# EPICS substitutions: ssaApp/Db/hlCommon.substitutions
# Common controls for cryomodule SSAs.
# Macros:
#   OUT: PV attribute
#   MASK: Bitmask to select which SSAs to control; e.g. 3 for SSAs 1 & 2, 15 for SSAs 1,2,3,4.
#   DLY: Delay between sequence steps

file "ssaCommonControls_4x.template" {
pattern
{       OUT, DLY}
{   PowerOn, 0.5}
{  PowerOff, 0.1}
{FaultReset, 0.5}
}
